TYPE stManipulatorPtpXYZ_DataRoot EXTENDS VortexBase.stVortexer:
STRUCT
END_STRUCT
END_TYPE

(* stored: Version 1.1.0.1
   DUT stManipulatorPtpXYZ_DataRoot: Id {86b7073d-19ad-0be4-0645-6a5850667066} *)
